TYPE ST_Monitoring_Module EXTENDS ST_Monitoring_Base :
STRUCT
	astMonitoring		: ARRAY[0..CONST.iMaxIdxMonitoring] OF ST_Data_Item;
	astMonitoringView	: ARRAY[0..CONST.iMaxIdxMonitoring] OF ST_Data_Item_String;
END_STRUCT
END_TYPE

(* stored: Version 1.1.0.1, ProductVersion 3.1.4024.12
   DUT ST_Monitoring_Module: Id {05882d8f-108a-43ac-a492-6a0bf00d86d3} *)
